{attribute 'qualified_only'}
VAR_GLOBAL
END_VAR

(* stored: Version 1.1.0.1, ProductVersion 3.1.4022.7
   GVL GVL_07_Alarm_Step_Motor: Id {57d70af5-1f83-4157-9edf-71f55e7cb7dd} *)
